FUNCTION_BLOCK RefactorRotatingArmControl (* Composite Function Block Type *)
  (* Standard: 61499-2 *)
  (* Version 0.0, 2/12/2018, Sandeep Patil, nxtControl GmbH, template *)
  PACKAGE Main;
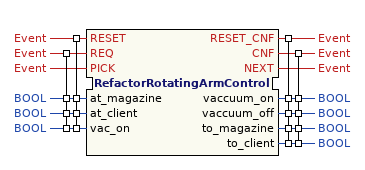
  EVENT_INPUT
    RESET WITH at_magazine, at_client, vac_on; (* Initialization Request *)
    REQ WITH at_magazine, at_client, vac_on; (* Normal Execution Request *)
    PICK;
  END_EVENT
  EVENT_OUTPUT
    RESET_CNF WITH vaccuum_on, vaccuum_off, to_magazine, to_client; (* Initialization Confirm *)
    CNF WITH vaccuum_on, vaccuum_off, to_magazine, to_client; (* Execution Confirmation *)
    NEXT;
  END_EVENT
  VAR_INPUT
    at_magazine : BOOL; (* Input event qualifier *)
    at_client : BOOL;
    vac_on : BOOL;
  END_VAR
  VAR_OUTPUT
    vaccuum_on : BOOL; (* Output event qualifier *)
    vaccuum_off : BOOL;
    to_magazine : BOOL;
    to_client : BOOL;
  END_VAR
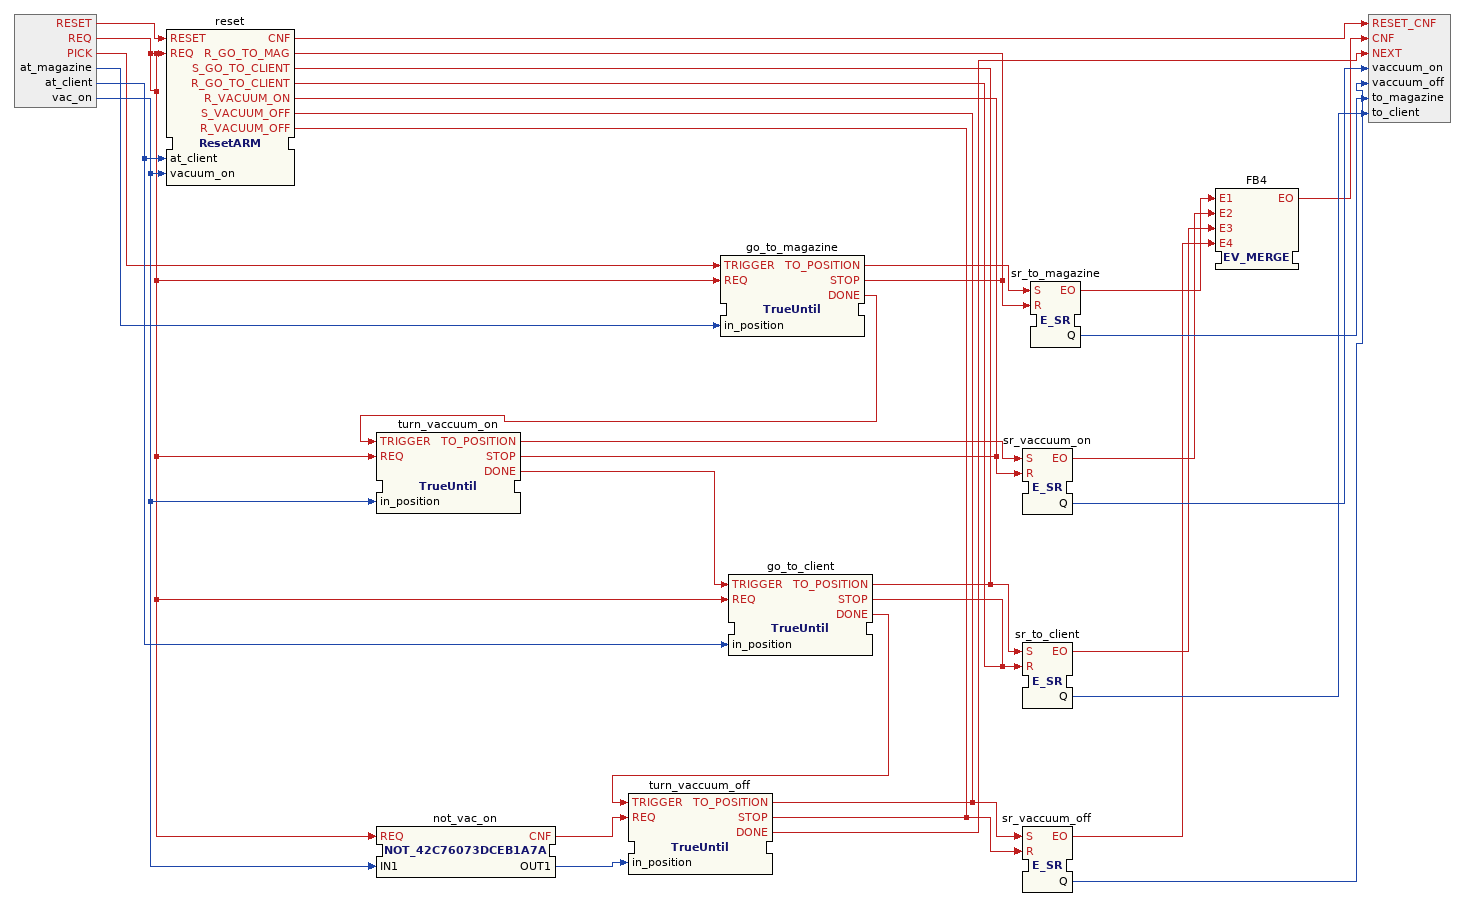
  FBS
    go_to_magazine : TrueUntil;
    turn_vaccuum_on : TrueUntil;
    go_to_client : TrueUntil;
    turn_vaccuum_off : TrueUntil;
    not_vac_on : NOT_42C76073DCEB1A7A; {SET_ATTRIBUTE(Configuration.GenericFBType.InterfaceParams, Runtime.Standard#CNT:=1;OUT${CNT$}:BOOL)}
    sr_vaccuum_on : E_SR;
    sr_vaccuum_off : E_SR;
    sr_to_magazine : E_SR;
    sr_to_client : E_SR;
    FB4 : EV_MERGE;
    reset : ResetARM;
  END_FBS
  EVENT_CONNECTIONS
    PICK TO go_to_magazine.TRIGGER;
    go_to_magazine.DONE TO turn_vaccuum_on.TRIGGER;
    turn_vaccuum_on.DONE TO go_to_client.TRIGGER;
    go_to_client.DONE TO turn_vaccuum_off.TRIGGER;
    not_vac_on.CNF TO turn_vaccuum_off.REQ;
    turn_vaccuum_off.DONE TO NEXT;
    REQ TO go_to_magazine.REQ;
    REQ TO turn_vaccuum_on.REQ;
    REQ TO go_to_client.REQ;
    REQ TO not_vac_on.REQ;
    turn_vaccuum_on.TO_POSITION TO sr_vaccuum_on.S;
    turn_vaccuum_on.STOP TO sr_vaccuum_on.R;
    go_to_magazine.TO_POSITION TO sr_to_magazine.S;
    go_to_magazine.STOP TO sr_to_magazine.R;
    go_to_client.TO_POSITION TO sr_to_client.S;
    go_to_client.STOP TO sr_to_client.R;
    turn_vaccuum_off.TO_POSITION TO sr_vaccuum_off.S;
    turn_vaccuum_off.STOP TO sr_vaccuum_off.R;
    RESET TO reset.RESET;
    reset.CNF TO RESET_CNF;
    sr_to_magazine.EO TO FB4.E1;
    sr_vaccuum_on.EO TO FB4.E2;
    sr_to_client.EO TO FB4.E3;
    sr_vaccuum_off.EO TO FB4.E4;
    FB4.EO TO CNF;
    reset.R_GO_TO_MAG TO sr_to_magazine.R;
    reset.S_GO_TO_CLIENT TO sr_to_client.S;
    reset.R_VACUUM_ON TO sr_vaccuum_on.R;
    reset.S_VACUUM_OFF TO sr_vaccuum_off.S;
    reset.R_GO_TO_CLIENT TO sr_to_client.R;
    reset.R_VACUUM_OFF TO sr_vaccuum_off.R;
    REQ TO reset.REQ;
  END_CONNECTIONS
  DATA_CONNECTIONS
    vac_on TO turn_vaccuum_on.in_position;
    at_client TO go_to_client.in_position;
    at_magazine TO go_to_magazine.in_position;
    vac_on TO not_vac_on.IN1;
    not_vac_on.OUT1 TO turn_vaccuum_off.in_position;
    sr_vaccuum_on.Q TO vaccuum_on;
    sr_vaccuum_off.Q TO vaccuum_off;
    sr_to_magazine.Q TO to_magazine;
    sr_to_client.Q TO to_client;
    vac_on TO reset.vacuum_on;
    at_client TO reset.at_client;
  END_CONNECTIONS
END_FUNCTION_BLOCK
